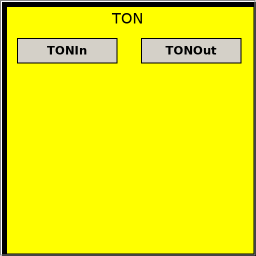
VISUALIZATION V_PH_TON  // 256x256
VAR_INPUT
	stSafetyTON			:ST_SAFETY_FBTON;
END_VAR
    Rectangle (2,2 256x256), colour toggle: stSafetyTON.bGeneralError
    Label (5,6 246x25), "TON"
    RoundedRectangle (17,38 100x25), "TONIn", colour toggle: stSafetyTON.uStatus.stStatusWords.wInputs.8
    RoundedRectangle (141,38 100x25), "TONOut", colour toggle: stSafetyTON.uStatus.stStatusWords.wOutputs.1
    Textfield (17,226 234x25), text list: 'TL_FbStateTimer', text index: stSafetyTON.eState
END_VISUALIZATION

(* stored: Version 1.1.0.1, ProductVersion 3.1.4024.4
   Visu V_PH_TON: Id {33272892-3df1-4bd8-bdd8-3f3c133a1002} *)
